TYPE ST_AxisConfig_back :
STRUCT

    ///////Axis Parameters//////
    fOverride           :   LREAL := 100;   //Controller override %
    fVelocity           :   LREAL;          //Velocity must be specified, no default used
    fAcceleration       :   LREAL;          //Not all FBs use, need to change this, 0 is NC default
    fDeceleration       :   LREAL;
    fPosition           :   LREAL;          //Used for absolute positioning
    fHomePosition       :   LREAL;          //Used to home to a value other than 0
    nHomeSeq            :   UINT;           //Homing sequence to perform
    eRestorePosition    :   RestorePosition;
    //Restore position of incremental axis after loss of power to the CPU, 0=don't restore, 1=restore but don't home, 2=restore and home

END_STRUCT
END_TYPE

(* stored: Version 1.1.0.1, ProductVersion 3.1.4024.6
   DUT ST_AxisConfig_back: Id {e00fe310-8ff8-452a-800a-823efa83b1a3} *)
